// TIA Portal V17 export
// export: Created 2022-07-28T18:03:17.2127763Z, ExportSetting None, DisplayName Totally Integrated Automation Portal, DisplayVersion V17, DisplayName TIA Portal Openness, DisplayVersion V17, DisplayName TIA Portal Teamcenter Gateway, DisplayVersion V17, DisplayName TIA Portal Version Control Interface, DisplayVersion V17, DisplayName TIA Portal Test Suite Advanced, DisplayVersion V17, DisplayName SINAMICS Startdrive Advanced, DisplayVersion V17, DisplayName SINAMICS DCC, DisplayVersion V17, DisplayName SINAMICS Startdrive G130, G150, S120, S150, SINAMICS MV, S210, DisplayVersion V17, DisplayName SINAMICS Startdrive G110M, G120, G120C, G120D, G120P, G115D, DisplayVersion V17, DisplayName STEP 7 Professional, DisplayVersion V17, DisplayName SIMATIC Energy Suite, DisplayVersion V17, DisplayName STEP 7 CFC, DisplayVersion V17, DisplayName STEP 7 Safety, DisplayVersion V17, DisplayName WinCC Advanced / Unified PC, DisplayVersion V17, DisplayName SIMATIC Visualization Architect, DisplayVersion V17
TYPE "_Inverter_352Tel_Recv"
   STRUCT
      STW : "_Inverter_352Tel_STW_Bits";   // Status word
      Running : Bool;   // 1 = running in any dirrection
      RunningForward : Bool;   // 1 = running in forward dirrection (act>0.0)
      RunningReverse : Bool;   // 1 = running in reverse dirrection (act<0.0)
      r_ActualSpeed : Real := 0.0;   // Actual speed, % from P2000
      r_ActualCurrent : Real := 0.0;   // Actual current, % from P2002
      r_ActualTorque : Real := 0.0;   // Actual torque, % from P2003
      w_Warning : Word;   // ID of actual warning
      w_Fault : Word;   // ID of actual fault
   END_STRUCT;
END_TYPE
